// User defined boolean value extension.
// > Contains additional parameters.
FUNCTION_BLOCK FB_UDef_BValEx EXTENDS FB_BA_BV_OP
VAR_INPUT CONSTANT
	{region 'Variable Parameters'}
		{attribute 'BaParam.Title.DE' := 'Erwarteter Wert'}
		{attribute 'BaParam.Title.EN' := 'Expected value'}
		{attribute 'BaParam.Access.Read' := 'Guest'}
		{attribute 'BaParam.Access.Write' := 'Advanced'}
		bExpected : BOOL;
	{endregion}
END_VAR
VAR_OUTPUT
	{attribute 'BaParam.Title.DE' := 'Übereinstimmend'}
	{attribute 'BaParam.Title.EN' := 'Matched'}
	{attribute 'BaParam.Access.Read' := 'Guest'}
	bMatch : BOOL;
END_VAR

SUPER^();

bMatch := (bPresentValue = bExpected);

END_FUNCTION_BLOCK

(* stored: Version 1.1.0.1, ProductVersion 3.1.4024.11
   POU FB_UDef_BValEx: Id {a6978dd8-3c4e-431f-8ccf-5ebd35a43806}, SpecialFunc None *)
